TYPE ST_ServoList :
STRUCT
	TableAxis : ST_ServoParaBasic;
END_STRUCT
END_TYPE

(* stored: Version 1.1.0.1, ProductVersion 3.1.4024.13
   DUT ST_ServoList: Id {88e8735f-6e17-4642-8496-f1ff0f110fae} *)
